Omron Sysmac Studio project PC_Envia_PLC_Recibe_1 (Sysmac Studio 1.23.0.14, StandardProject)

# Controller new_Controller_0: NX1P2-1040DT1 version 1.18
Task PrimaryTask (priority 4, period or condition 2000): Programa0

VAR_GLOBAL
    Mi_Puerto : _sDEVICE_PORT;
END_VAR
VAR_GLOBAL CONSTANT
    Mi_Modulo485 : _sOPTBOARD_ID := (SlotNo := 2, IPAdr := [5(16#0)]);
END_VAR
VAR_GLOBAL
    MiBufKind : _eSERIAL_BUF_KIND := _BUF_SENDRCV;
    Sensibilidad_Rcv : _sSERIAL_CFG;
    Orden_Leer : BOOL;
    Dato : ARRAY[0..1] OF BYTE;
    Valor_Sal_0_ON : ARRAY[0..1] OF BYTE := [16#34, 16#F2];
    Valor_Sal_0_OFF : ARRAY[0..1] OF BYTE := [16#25, 16#31];
    Sal_0 : BOOL;  (* at BuiltInIO://cpu/#0/Output_Bit_00 *)
END_VAR

PROGRAM Programa0
VAR
    NX_SerialBufClear_Instance : NX_SerialBufClear;
    NX_SerialBufClear_Instance1 : NX_SerialBufClear;
    NX_SerialRcv_Instance1 : NX_SerialRcv;
    NX_SerialBufClear_Instance2 : NX_SerialBufClear;
END_VAR
VAR_EXTERNAL
    Mi_Puerto : _sDEVICE_PORT;
END_VAR
VAR_EXTERNAL CONSTANT
    Mi_Modulo485 : _sOPTBOARD_ID;
END_VAR
VAR_EXTERNAL
    Sensibilidad_Rcv : _sSERIAL_CFG;
    MiBufKind : _eSERIAL_BUF_KIND;
    Orden_Leer : BOOL;
    Dato : ARRAY[0..1] OF BYTE;
    Valor_Sal_0_ON : ARRAY[0..1] OF BYTE;
    Sal_0 : BOOL;
    Valor_Sal_0_OFF : ARRAY[0..1] OF BYTE;
END_VAR
VAR
    _e1 : F_TRIG;
    _e2 : R_TRIG;
END_VAR

(* Section Recepción: ladder, written here as Structured Text *)

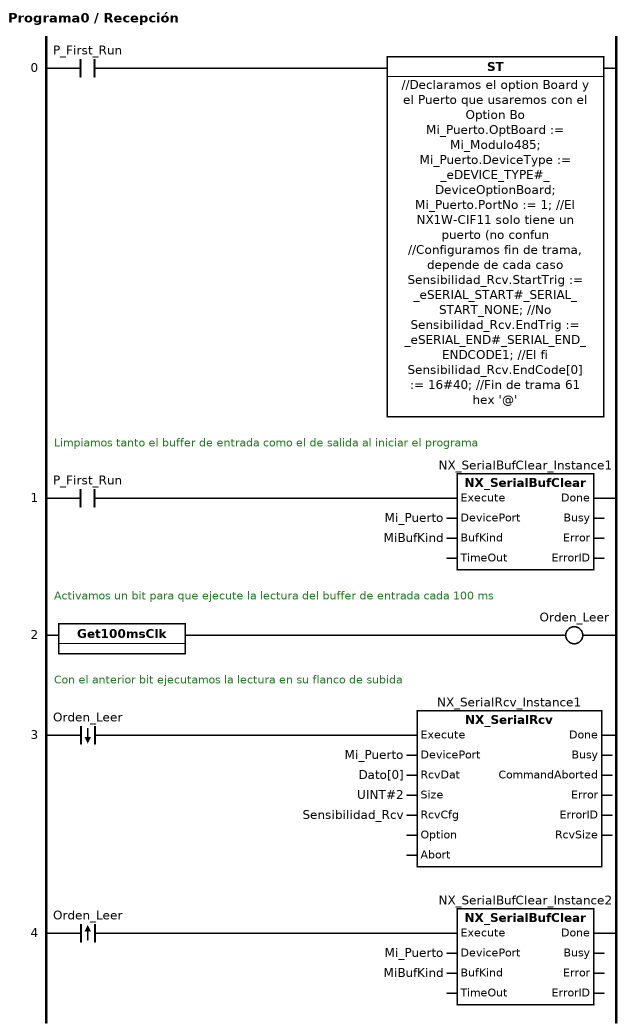
(* Rung 0 *)
IF P_First_Run THEN
    //Declaramos el option Board y el Puerto que usaremos con el Option Board anterior.
    Mi_Puerto.OptBoard := Mi_Modulo485;
    Mi_Puerto.DeviceType := _eDEVICE_TYPE#_DeviceOptionBoard;
    Mi_Puerto.PortNo := 1; //El NX1W-CIF11 solo tiene un puerto (no confundir con el slot donde está el módulo)
    
    //Configuramos fin de trama, depende de cada caso
    Sensibilidad_Rcv.StartTrig := _eSERIAL_START#_SERIAL_START_NONE; //No hay código de inicio
    Sensibilidad_Rcv.EndTrig := _eSERIAL_END#_SERIAL_END_ENDCODE1; //El final es marcado por cualquier byte
    Sensibilidad_Rcv.EndCode[0] := 16#40; //Fin de trama 61 hex '@'
END_IF;
(* Rung 1: Limpiamos tanto el buffer de entrada como el de salida al iniciar el programa *)
NX_SerialBufClear_Instance1(Execute := P_First_Run, DevicePort := Mi_Puerto, BufKind := MiBufKind);
(* Rung 2: Activamos un bit para que ejecute la lectura del buffer de entrada cada 100 ms *)
Orden_Leer := Get100msClk();
(* Rung 3: Con el anterior bit ejecutamos la lectura en su flanco de subida *)
_e1(CLK := Orden_Leer);
NX_SerialRcv_Instance1(Execute := _e1.Q, DevicePort := Mi_Puerto, RcvDat := Dato[0], Size := UINT#2, RcvCfg := Sensibilidad_Rcv);
(* Rung 4 *)
_e2(CLK := Orden_Leer);
NX_SerialBufClear_Instance2(Execute := _e2.Q, DevicePort := Mi_Puerto, BufKind := MiBufKind);

(* Section Salida: ladder, written here as Structured Text *)

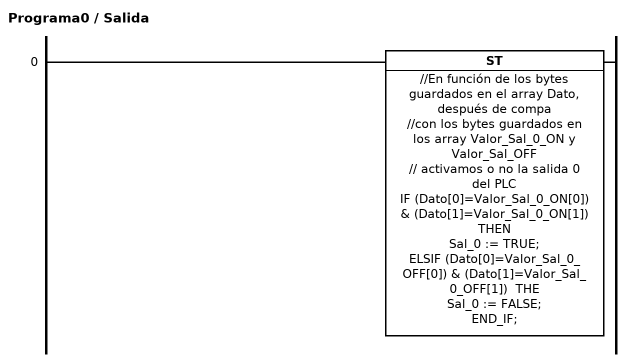
(* Rung 0 *)
//En función de los bytes guardados en el array Dato, después de compararlos
//con los bytes guardados en los array Valor_Sal_0_ON y Valor_Sal_OFF
// activamos o no la salida 0 del PLC
IF (Dato[0]=Valor_Sal_0_ON[0]) & (Dato[1]=Valor_Sal_0_ON[1]) THEN
    Sal_0 := TRUE;
ELSIF (Dato[0]=Valor_Sal_0_OFF[0]) & (Dato[1]=Valor_Sal_0_OFF[1])  THEN
	Sal_0 := FALSE;
END_IF;
END_PROGRAM